FUNCTION_BLOCK EtherNetIPDeviceBase
VAR_INPUT
END_VAR
VAR_OUTPUT
END_VAR
VAR
	State AT%i* : UINT;
END_VAR

END_FUNCTION_BLOCK

(* stored: Version 1.1.0.1, ProductVersion 3.1.4024.11
   POU EtherNetIPDeviceBase: Id {04ea0fee-aaad-4194-8290-79848d5bf3ea}, SpecialFunc None *)
